(* Logix 5000 project; controller PLC_IA vendor 1 type 14 code 15 rev 20.11; software revision 20.05 *)

TASK MainTask (continuous, watchdog 500 ms) : MainProgram

MODULES
   Local : vendor 1 type 14 code 15 (SoftLogixController 1, rev 20.11)
END_MODULES

VAR_GLOBAL   (* controller tags *)
   ATRASO_SENSOR : REAL := 1000.0;
   CONST_TEMPO : REAL := 15.0;
   DELTA_T : REAL := 0.01;
   ERRO : REAL := 3.9972687;
   FATOR_CONSUMO : REAL := 100.0;
   FLUXO_VAPOR : REAL := 90.0;
   FUZZY_LOOP : FBD_TIMER := (TimerEnable := 1, PRE := 40, ACC := 20, EN := 1, TT := 1);
   FUZZY_ON : BOOL := 1;
   KP : REAL := 3.0;
   KP_MANUAL : REAL := 7.0;
   KP_MAX : REAL := 10.0;
   KP_MIN : REAL := 3.0;
   LIGA_SISTEMA : BOOL := 1;
   MV : REAL := 53.90078;
   P_MAX : REAL := 250.0;
   PV : REAL := 171.15842;
   SP : REAL := 175.0;
   T_AMOST_PID : REAL := 50.0;
   T_LOOP_SISTEMA : REAL := 10.0;
   TAU : REAL := 1.5;
   TD : REAL := 4.274473;
   TD_MANUAL : REAL := 1.0;
   TD_MAX : REAL := 5.0;
   TD_MIN : REAL := 1.0;
   TI : REAL := 5.0;
   TI_INV : REAL := 0.22324193;
   TI_MANUAL : REAL := 3.0;
   TI_MAX : REAL := 5.0;
   TI_MIN : REAL := 0.5;
   VAZAMENTO : REAL;
END_VAR

PROGRAM FUZZY   (* main routine PRINCIPAL *)
VAR
   ACC_DERIVADA : REAL := 0.7598929;
   ACC_DESVIOS_QUADRADO : REAL := 0.0010012466;
   ACC_ERRO : REAL;
   AMOSTRAGEM : FBD_TIMER := (TimerEnable := 1, PRE := 20);
   BUFFER_CIRCULAR : BOOL := 1;
   CONTAGEM : DINT := 46;
   DERIVADA_ALTA : REAL := 0.00604254;
   DERIVADA_BAIXA : REAL := 0.0015563883;
   DERIVADA_FILTRADA : REAL := 0.0023156737;
   DERIVADA_MEDIA : REAL := 0.0037994643;
   DERIVADAS : REAL[5] := ([2] := 0.008644867, [4] := 0.008800507);
   DESVIO : REAL := -0.0014837906;
   DESVIO_PADRAO : REAL := 0.002243076;
   ERRO_ALTO : REAL := 17.5;
   ERRO_ANTERIOR : REAL := 3.9972687;
   ERRO_BAIXO : REAL := 0.17500001;
   ERRO_FILTRADO : REAL := 4.1489806;
   ERRO_MEDIO : REAL := 1.75;
   ERROS : REAL[5] := ([0] := 3.9972687, [1] := 4.346176, [2] := 4.173279, [3] := 4.173279, [4] := 3.9972687);
   EXECUCAO : DINT;
   FILTRAGEM : FBD_TIMER := (TimerEnable := 1, PRE := 20, EN := 1, TT := 1);
   FUZZ_KP : REAL[3] := ([0] := 0.43700165, [2] := 0.1552568);
   FUZZ_TD : REAL[3] := ([0] := 0.1552568, [1] := 0.4403919, [2] := 0.5596081);
   FUZZ_TI : REAL[3] := ([0] := 0.43700165, [1] := 0.8447432, [2] := 0.5596081);
   FUZZY_TIME : REAL := 40.0;
   KP_ALTO : REAL := 10.0;
   KP_BAIXO : REAL := 3.0;
   KP_MEDIO : REAL := 6.5;
   MENOR_VALOR : REAL;
   PERTI_DERIVADA : REAL[3] := ([1] := 0.4403919, [2] := 0.5596081);
   PERTI_ERRO : REAL[3] := ([1] := 0.8447432, [2] := 0.1552568);
   POSICAO : DINT := 1;
   PRIMEIRA_EXECUCAO : BOOL;
   T_AMOSTRAGEM : FBD_TIMER := (Reset := 1);
   TAMANHO_BUFFER : REAL := 200.0;
   TD_ALTO : REAL := 5.0;
   TD_BAIXO : REAL := 1.0;
   TD_MEDIO : REAL := 3.0;
   TEMPO_AMOSTRAGEM : REAL := 20.0;
   TI_ALTO : REAL := 5.0;
   TI_BAIXO : REAL := 0.5;
   TI_MEDIO : REAL := 2.75;
   TIME_FILTRAGEM : REAL := 20.0;
   ULTIMA_DERIVADA : REAL;
   VARIANCIA : REAL := 5.03139e-06;
   VETOR_DERIVADAS : REAL[201] := ([0] := 0.0037889606, [1] := 0.0020592753, [2] := 0.00418396, [3] := 0.0020858257, [4] := 0.0060199993, [5] := 0.003966878, [6] := 0.0034370932, [7] := 0.005819702, [8] := 0.0041832477, [9] := 0.0057259626, [10] := 0.0025300598, [11] := 0.008794352, [12] := 0.005414327, [13] := 0.004825694, [14] := 0.008985087, [15] := 0.006632945, [16] := 0.007867635, [17] := 0.0036768594, [18] := 0.0064361067, [19] := 0.0027026369, [20] := 0.0034643046, [21] := 0.0013593547, [22] := 0.0011015829, [23] := 0.0010068257, [24] := 0.00049591064, [25] := 0.0017445373, [26] := 0.0017635092, [27] := 0.0010932413, [28] := 0.0035477194, [29] := 0.0020349121, [30] := 0.0050069173, [31] := 0.002079061, [32] := 0.0069529214, [33] := 0.0042039487, [34] := 0.00426946, [35] := 0.005052897, [36] := 0.0044214376, [37] := 0.0038611856, [38] := 0.0016247558, [39] := 0.0046980795, [40] := 0.0026897178, [41] := 0.0025284833, [42] := 0.0047458396, [43] := 0.0031422423, [44] := 0.0050496925, [45] := 0.0023156737, [46] := 0.00046005248, [47] := 0.00038441975, [48] := 0.00032608034, [49] := 0.00015319824, [50] := 0.0007211812, [51] := 0.00089324947, [52] := 0.0004510498, [53] := 0.002618103, [54] := 0.0012327576, [55] := 0.0043327333, [56] := 0.0018105062, [57] := 0.005733185, [58] := 0.0038183595, [59] := 0.0038228354,
        [60] := 0.0052285767, [61] := 0.0037962343, [62] := 0.0052091475, [63] := 0.0023093158, [64] := 0.006299642, [65] := 0.0037178549, [66] := 0.0037252808, [67] := 0.0050693764, [68] := 0.0036811319, [69] := 0.005033366, [70] := 0.0022351076, [71] := 0.006123454, [72] := 0.003578135, [73] := 0.0036023457, [74] := 0.004944407, [75] := 0.0035803223, [76] := 0.00487381, [77] := 0.002181193, [78] := 0.0059391274, [79] := 0.0034865316, [80] := 0.0034903463, [81] := 0.0047751362, [82] := 0.0034667968, [83] := 0.004758555, [84] := 0.002109375, [85] := 0.0057554627, [86] := 0.0033972675, [87] := 0.0034038797, [88] := 0.004633484, [89] := 0.003364156, [90] := 0.00460083, [91] := 0.0020432028, [92] := 0.0055985004, [93] := 0.0032713318, [94] := 0.0032933552, [95] := 0.0045218403, [96] := 0.0032740275, [97] := 0.004457957, [98] := 0.0019950867, [99] := 0.0054330444, [100] := 0.0031900024, [101] := 0.0031932069, [102] := 0.004369812, [103] := 0.0031721496, [104] := 0.004355367, [105] := 0.0019306437, [106] := 0.0052687074, [107] := 0.0031103517, [108] := 0.003116099, [109] := 0.004243113, [110] := 0.0030804952, [111] := 0.0042140707, [112] := 0.0018713379, [113] := 0.005128072, [114] := 0.002996877, [115] := 0.0030169168, [116] := 0.0041429647, [117] := 0.0029994203, [118] := 0.0040854393, [119] := 0.0018282572,
        [120] := 0.004979502, [121] := 0.002924245, [122] := 0.0029269918, [123] := 0.004005992, [124] := 0.002907969, [125] := 0.0039934795, [126] := 0.0017700704, [127] := 0.0044295248, [128] := 0.0021709695, [129] := 0.0025767009, [130] := 0.0014201864, [131] := 0.0017451985, [132] := 0.0012846374, [133] := 0.00026168823, [134] := 0.0024367778, [135] := 0.0021867373, [136] := 0.0017131043, [137] := 0.0052009076, [138] := 0.0030574545, [139] := 0.006877899, [140] := 0.0029870605, [141] := 0.009012044, [142] := 0.005469309, [143] := 0.0057130945, [144] := 0.0072477725, [145] := 0.0054625957, [146] := 0.007619018, [147] := 0.003203481, [148] := 0.009398296, [149] := 0.005638784, [150] := 0.005854645, [151] := 0.007651062, [152] := 0.0056430562, [153] := 0.008111725, [154] := 0.0034550477, [155] := 0.009210052, [156] := 0.0057525635, [157] := 0.0058767702, [158] := 0.008184764, [159] := 0.005391744, [160] := 0.00840266, [161] := 0.003948822, [162] := 0.008733826, [163] := 0.004367625, [164] := 0.005135396, [165] := 0.0042689512, [166] := 0.0032692973, [167] := 0.0043944293, [168] := 0.0018687438, [169] := 0.006122894, [170] := 0.004126994, [171] := 0.0038800559, [172] := 0.0067077638, [173] := 0.004504191, [174] := 0.007554728, [175] := 0.0033129374, [176] := 0.008668976, [177] := 0.004777832, [178] := 0.0053255716, [179] := 0.0052858484,
        [180] := 0.004243876, [181] := 0.0037680052, [182] := 0.0018651835, [183] := 0.0036832173, [184] := 0.0015258789, [185] := 0.0017882792, [186] := 0.000923818, [187] := 0.0010198465, [188] := 0.00053400674, [189] := 0.00016108195, [190] := 0.0007420858, [191] := 0.00032419842, [192] := 0.00037216189, [193] := 0.0015240987, [194] := 0.0007048544, [195] := 0.0016716511, [196] := 0.0009288025, [197] := 0.0025672913, [198] := 0.0018614196, [199] := 0.0015527343, [200] := 0.03885905);
   VETOR_DESVIOS : REAL[201] := ([0] := 2.9573382e-06, [1] := 2.5091268e-07, [2] := 1.5205011e-06, [3] := 7.661391e-07, [4] := 1.5119083e-06, [5] := 7.2051694e-06, [6] := 3.784602e-07, [7] := 6.891656e-09, [8] := 5.9700624e-06, [9] := 6.488707e-07, [10] := 5.4367933e-06, [11] := 7.475152e-07, [12] := 2.885194e-05, [13] := 3.9043834e-06, [14] := 1.8993056e-06, [15] := 3.0242056e-05, [16] := 9.806415e-06, [17] := 1.8807697e-05, [18] := 1.8989514e-08, [19] := 8.281695e-06, [20] := 7.388706e-07, [21] := 1.0648864e-08, [22] := 4.88189e-06, [23] := 6.0449424e-06, [24] := 6.505347e-06, [25] := 9.338245e-06, [26] := 3.2610042e-06, [27] := 3.197212e-06, [28] := 6.0241664e-06, [29] := 1.8111357e-10, [30] := 2.3277132e-06, [31] := 2.0372106e-06, [32] := 2.2642676e-06, [33] := 1.1167069e-05, [34] := 3.3333185e-07, [35] := 3.946825e-07, [36] := 1.9304443e-06, [37] := 5.5261563e-07, [38] := 2.8178214e-08, [39] := 4.2948723e-06, [40] := 9.648893e-07, [41] := 1.072789e-06, [42] := 1.4534289e-06, [43] := 9.799563e-07, [44] := 3.9057537e-07, [45] := 1.58615e-06, [46] := 8.007315e-06, [47] := 8.10455e-06, [48] := 8.487863e-06, [49] := 8.782421e-06, [50] := 9.7864795e-06, [51] := 6.4863684e-06, [52] := 5.606348e-06, [53] := 7.79847e-06, [54] := 3.9699964e-07, [55] := 3.997394e-06, [56] := 1.1974279e-06, [57] := 2.023872e-06, [58] := 6.2132062e-06, [59] := 3.2789654e-07,
        [60] := 3.4131332e-07, [61] := 3.900039e-06, [62] := 3.1043325e-07, [63] := 3.865559e-06, [64] := 8.5381527e-07, [65] := 9.403526e-06, [66] := 2.388203e-07, [67] := 2.6127444e-07, [68] := 3.4021562e-06, [69] := 2.2981268e-07, [70] := 3.3539004e-06, [71] := 9.082978e-07, [72] := 8.640061e-06, [73] := 1.610975e-07, [74] := 1.9430595e-07, [75] := 3.144376e-06, [76] := 1.8326233e-07, [77] := 2.9420125e-06, [78] := 9.357414e-07, [79] := 7.683639e-06, [80] := 9.994215e-08, [81] := 9.622623e-08, [82] := 2.4721726e-06, [83] := 6.588723e-08, [84] := 2.3537712e-06, [85] := 1.2501492e-06, [86] := 6.356949e-06, [87] := 2.5232172e-08, [88] := 3.0898907e-08, [89] := 1.9450006e-06, [90] := 2.0357055e-08, [91] := 1.890251e-06, [92] := 1.3742845e-06, [93] := 5.6442605e-06, [94] := 2.4645186e-09, [95] := 5.3044302e-09, [96] := 1.6544536e-06, [97] := 1.5958361e-09, [98] := 1.4656536e-06, [99] := 1.5662874e-06, [100] := 4.6900473e-06, [101] := 7.498061e-09, [102] := 9.312055e-09, [103] := 1.1222714e-06, [104] := 2.2385308e-08, [105] := 1.0286437e-06, [106] := 2.0112932e-06, [107] := 3.609533e-06, [108] := 7.2895325e-08, [109] := 7.4481704e-08, [110] := 6.990904e-07, [111] := 1.1010914e-07, [112] := 6.207139e-07, [113] := 2.427668e-06, [114] := 2.845061e-06, [115] := 2.0363854e-07, [116] := 1.8261623e-07, [117] := 4.705508e-07, [118] := 1.9731706e-07, [119] := 4.108834e-07,
        [120] := 2.5830077e-06, [121] := 2.4127462e-06, [122] := 2.441865e-07, [123] := 2.1766195e-07, [124] := 3.7180462e-07, [125] := 2.0217527e-07, [126] := 4.2309293e-07, [127] := 2.3991495e-06, [128] := 1.3035926e-06, [129] := 1.1903454e-06, [130] := 4.0863705e-07, [131] := 3.158271e-06, [132] := 1.917442e-06, [133] := 3.253678e-06, [134] := 7.737029e-06, [135] := 2.980862e-07, [136] := 5.727842e-07, [137] := 1.3515066e-06, [138] := 5.4450447e-06, [139] := 7.169536e-08, [140] := 1.6864713e-05, [141] := 6.5627745e-08, [142] := 3.9622384e-05, [143] := 7.695371e-06, [144] := 9.224776e-06, [145] := 2.0757028e-05, [146] := 7.797909e-06, [147] := 2.4361989e-05, [148] := 2.8252762e-07, [149] := 4.498373e-05, [150] := 8.652641e-06, [151] := 9.921689e-06, [152] := 2.4187766e-05, [153] := 8.438927e-06, [154] := 2.8561488e-05, [155] := 4.6599374e-07, [156] := 4.1015617e-05, [157] := 8.573145e-06, [158] := 9.207904e-06, [159] := 2.8160855e-05, [160] := 6.2536906e-06, [161] := 3.0007364e-05, [162] := 1.0253484e-06, [163] := 3.3237407e-05, [164] := 1.9191352e-06, [165] := 4.571872e-06, [166] := 1.575745e-06, [167] := 6.3512125e-08, [168] := 1.8560517e-06, [169] := 1.3580159e-06, [170] := 9.41174e-06, [171] := 1.1200739e-06, [172] := 6.4198497e-07, [173] := 1.2957162e-05, [174] := 1.9173199e-06, [175] := 1.9393981e-05, [176] := 2.3088429e-08, [177] := 2.995802e-05, [178] := 2.4483259e-06, [179] := 4.3870746e-06,
        [180] := 4.1300164e-06, [181] := 9.595819e-07, [182] := 2.411631e-07, [183] := 2.0017692e-06, [184] := 1.5463954e-07, [185] := 3.1172626e-06, [186] := 2.2611748e-06, [187] := 5.612499e-06, [188] := 5.1435136e-06, [189] := 7.565125e-06, [190] := 9.723186e-06, [191] := 6.414435e-06, [192] := 8.680194e-06, [193] := 8.363685e-06, [194] := 3.0417334e-06, [195] := 6.5379736e-06, [196] := 2.536733e-06, [197] := 5.449436e-06, [198] := 4.911451e-07, [199] := 1.9887643e-06);
   VETOR_ERRO : REAL[201];
END_VAR

ROUTINE FUZZY   (* structured text *)
   ////////////////////////////////////////////////////////////////////////////////////////
   //						FILTRAGEM DAS VARIAVES DE ENTRADA
   ////////////////////////////////////////////////////////////////////////////////////////
   
   
   
   //TIMER DE FILTRAGEM
   TONR(FILTRAGEM);
   TIME_FILTRAGEM			:= T_LOOP_SISTEMA*2;
   FILTRAGEM.PRE 			:= TIME_FILTRAGEM;
   FILTRAGEM.ENABLEIN 		:= 1;
   FILTRAGEM.RESET 		:= 0;
   FILTRAGEM.TIMERENABLE	:= 1;
   
   
   //DISPARO DO TIMER
   IF FILTRAGEM.DN THEN
   
   	//RESETA O TIMER
   	FILTRAGEM.RESET := 1;
   
   	//SALVA O ERRO ABSOLUTO ATUAL
   	ERROS[POSICAO]:= ABS(ERRO);
   
   	//SALVA A DERIVADA ABSOLUTA ATUAL
   	DERIVADAS[POSICAO] := ABS((ERROS[POSICAO] - ERRO_ANTERIOR)/TIME_FILTRAGEM);
   
   	//SALVA O ULTIMO ERRO
   	ERRO_ANTERIOR := ERROS[POSICAO];
   
   	//NAO DEIXA TIRAR A MEDIA PONDERADA ENQUANTO O BUFFER NAO ESTA COMPLETAMENTE CHEIO
   	IF NOT(PRIMEIRA_EXECUCAO) THEN
   
   		//ERRO DE ENTRADA DO FUZZIFICADOR
   		ERRO_FILTRADO := (ERROS[(POSICAO) MOD 5]*5 + ERROS[(POSICAO+1) MOD 5]*4 + ERROS[(POSICAO+2) MOD 5]*3
   					+ ERROS[(POSICAO+3) MOD 5]*2 + ERROS[(POSICAO+4) MOD 5])/15;
   
   		//DERIVADA DE ENTRADA DO FUZZIFICADOR
   		DERIVADA_FILTRADA := (DERIVADAS[(POSICAO) MOD 5]*5 + DERIVADAS[(POSICAO+1) MOD 5]*4 + DERIVADAS[(POSICAO+2) MOD 5]*3
   					+ DERIVADAS[(POSICAO+3) MOD 5]*2 + DERIVADAS[(POSICAO+4) MOD 5])/15;
   	ELSE
   
   		//CONTA A QUANTIDADE DE POSICOES CHEIAS NO BUFFER
   		EXECUCAO := EXECUCAO + 1;
   
   		//SE ENCHEU FLIPA O BIT QUE DEIXA TIRAR A MEDIA
   		IF EXECUCAO > 4 THEN
   			EXECUCAO 		 	:= 0;
   			PRIMEIRA_EXECUCAO 	:= 0;
   		END_IF;
   
   	END_IF;
   
   
   	//INCREMENTA O BUFFER CIRCULAR
   	POSICAO := (POSICAO + 1) MOD 5;
   
   END_IF;
   
   
   
   
   ////////////////////////////////////////////////////////////////////////////////////////
   //		DEFININDO OS REFERENCIAIS DE ERRO
   
   ERRO_BAIXO := 0.001*SP;
   ERRO_MEDIO := 0.05*SP;
   ERRO_ALTO  := 0.15*SP;
   
   
   ////////////////////////////////////////////////////////////////////////////////////////
   //		ANALIZANDO AS ESTATISTICAS DAS ULTIMAS 200 VARIACOES DO ERRO (DERIVADA)
   
   
   //TIMER DE AMOSTRAGEM
   TONR(AMOSTRAGEM);
   TEMPO_AMOSTRAGEM		:= T_LOOP_SISTEMA*2;
   AMOSTRAGEM.PRE 			:= TEMPO_AMOSTRAGEM;
   AMOSTRAGEM.ENABLEIN 	:= 1;
   AMOSTRAGEM.TIMERENABLE 	:= 1;
   AMOSTRAGEM.RESET 		:= 0;
   
   IF AMOSTRAGEM.DN THEN
   
   	AMOSTRAGEM.RESET 		:= 1;
   	AMOSTRAGEM.TIMERENABLE 	:= 0;
   
   	//SE AUMENTAR MUITO ATRASA A RESPOSTA
   	TAMANHO_BUFFER := 200;
   
   	//LIGA O BUFFER CIRCULAR
   	IF BUFFER_CIRCULAR THEN
   
   		//RETIRA O ULTIMO VALOR DO VETOR DE DERIVADAS
   		ACC_DERIVADA := ACC_DERIVADA - VETOR_DERIVADAS[CONTAGEM];
   
   		//RETIRA O ULTIMO VALOR DO VETOR DE DESVIOS
   		ACC_DESVIOS_QUADRADO := ACC_DESVIOS_QUADRADO - VETOR_DESVIOS[CONTAGEM];
   
   	END_IF;
   
   	//ACUMULA OS K-ULTIMOS VALORES
   	ACC_DERIVADA:= ACC_DERIVADA + DERIVADA_FILTRADA;
   	ACC_DESVIOS_QUADRADO := ACC_DESVIOS_QUADRADO + DESVIO*DESVIO;
   
   	//SALVA A ULTIMA DERIVADA NO VETOR
   	VETOR_DERIVADAS[CONTAGEM] :=  DERIVADA_FILTRADA;
   
   	//SALVA O ULTIMO DESVIO NO VETOR
   	VETOR_DESVIOS[CONTAGEM] :=  DESVIO*DESVIO;
   
   	//INCREMENTA A CONTAGEM DE DERIVADAS
   	CONTAGEM := CONTAGEM + 1;
   
   	//SE A JANELA ENCHEU, LIGA O BUFFER CIRCULAR E VOLTA AO SEU INICIO
   	IF CONTAGEM > TAMANHO_BUFFER-1 THEN
   		BUFFER_CIRCULAR :=1;
   		CONTAGEM := 0;
   	END_IF;
   
   ////////////////////////////////////////////////////////////////////////////////////////
   //		DEFININDO OS REFERENCIAIS DA DERIVADA DO ERRO
   
   	//DERIVADA MEDIA (VARIAVEL DE REFERENCIA)
   	DERIVADA_MEDIA := ACC_DERIVADA/TAMANHO_BUFFER;
   
   	//DESVIO
   	DESVIO := DERIVADA_FILTRADA - DERIVADA_MEDIA;
   
   	//VARIANCIA COM UM GRAU DE LIBERDADE
   	VARIANCIA := ACC_DESVIOS_QUADRADO/(TAMANHO_BUFFER-1);
   
   	//DESVIO PADRAO
   	DESVIO_PADRAO := SQRT(VARIANCIA);
   
   	//VARIAVEIS DE REFERENCIA RESTANTES
   	DERIVADA_BAIXA := DERIVADA_MEDIA - DESVIO_PADRAO;
   	IF DERIVADA_BAIXA < 0 THEN
   		DERIVADA_BAIXA := 0;
   	END_IF;
   	DERIVADA_ALTA  := DERIVADA_MEDIA + DESVIO_PADRAO;
   
   END_IF;
   
   
   ////////////////////////////////////////////////////////////////////////////////////////
   //							CONTROLE DO ALGORITMO FUZZY
   ////////////////////////////////////////////////////////////////////////////////////////
   
   //TEMPO DE LOOP_FUZZY EM MILISSEGUNDOS
   //FUZZY_TIME := (TEMPO_AMOSTRAGEM*TAMANHO_BUFFER)/4;
   FUZZY_TIME := TEMPO_AMOSTRAGEM*2;
   
   //LIGA FUZZY
   IF FUZZY_ON THEN
   
   	//TIMER DE LOOP FUZZY
   	TONR(FUZZY_LOOP);
   	FUZZY_LOOP.PRE 			:= FUZZY_TIME;
   	FUZZY_LOOP.ENABLEIN 	:= 1;
   	FUZZY_LOOP.TIMERENABLE 	:= 1;
   	FUZZY_LOOP.RESET 		:= 0;
   
   ELSE
   	//RESET DO TEMPORIZADOR
   	FUZZY_LOOP.ENABLEIN 	:= 0;
   	FUZZY_LOOP.TIMERENABLE 	:= 0;
   	FUZZY_LOOP.RESET 		:= 1;
   	FUZZY_LOOP.DN			:= 0;
   
   	//RESET DAS VARIAVEIS DA MEDIA MOVEL
   	BUFFER_CIRCULAR			:= 0;
   	ACC_DERIVADA			:= 0;
   	ACC_DESVIOS_QUADRADO	:= 0;
   	CONTAGEM				:= 0;
   
   
   	//DESLIGA A AMOSTRAGEM ESTATISTICA
   	T_AMOSTRAGEM.TIMERENABLE 	:= 0;
   	T_AMOSTRAGEM.RESET 			:= 1;
   
   	//RETORNA AS VARIAVEIS SINTONIZADAS MANUALMENTE
   	KP := KP_MANUAL;
   	TI := TI_MANUAL;
   	TD := TD_MANUAL;
   
   	//RESET DA FILTRAGEM
   	POSICAO				:= 0;
   	ERRO_FILTRADO		:= 0;
   	DERIVADA_FILTRADA	:= 0;
   	PRIMEIRA_EXECUCAO 	:= 1;
   	EXECUCAO 		 	:= 0;
   
   
   END_IF;
   
   
   
   ////////////////////////////////////////////////////////////////////////////////////////
   //							INICIO DO ALGORITMO FUZZY
   ////////////////////////////////////////////////////////////////////////////////////////
   
   //TESTA SE O TIMER DE LOOP DISPAROU
   IF FUZZY_LOOP.DN THEN;
   
   
   ///////////////////////////////////////////////////////////////////////////////
   //			CALCULO DO VETOR DE PERTINENCIA DO ERRO
   
   	//CERTEZA DE QUE O ERRO EH BAIXO
   	IF ERRO_FILTRADO <= ERRO_BAIXO THEN
   		PERTI_ERRO[0] := 1;	//ERRO BAIXO
   		PERTI_ERRO[1] := 0;	//ERRO MEDIO
   		PERTI_ERRO[2] := 0;	//ERRO ALTO
   	ELSE
   
   		//CERTEZA DE QUE O ERRO EH ALTO
   		IF ERRO_FILTRADO >= ERRO_ALTO THEN
   			PERTI_ERRO[0] := 0;	//ERRO BAIXO
   			PERTI_ERRO[1] := 0;	//ERRO MEDIO
   			PERTI_ERRO[2] := 1;	//ERRO ALTO
   		ELSE
   
   			//MEIO TERMO
   			IF ERRO_FILTRADO < ERRO_MEDIO THEN
   
   				//SO PRA GARANTIR QUE NAO VAI DAR ERRO DE DIVISAO POR ZERO
   				IF ERRO_MEDIO <> ERRO_BAIXO THEN
   
   					//VAMOS CALCULAR PRIMEIRO O ERRO MEDIO
   					PERTI_ERRO[1] := (ERRO_FILTRADO-ERRO_BAIXO)/(ERRO_MEDIO-ERRO_BAIXO);
   
   				END_IF;
   
   				//ERRO BAIXO
   				PERTI_ERRO[0] := 1 - PERTI_ERRO[1];
   
   				//ERRO ALTO
   				PERTI_ERRO[2] := 0;
   
   			ELSE
   
   				//SO PRA GARANTIR QUE NAO VAI DAR ERRO DE DIVISAO POR ZERO
   				IF ERRO_MEDIO <> ERRO_ALTO THEN
   
   					//VAMOS CALCULAR PRIMEIRO O ERRO ALTO
   					PERTI_ERRO[2] := (ERRO_FILTRADO- ERRO_MEDIO)/(ERRO_ALTO-ERRO_MEDIO);
   
   				END_IF;
   
   				//PERTINENCIA DO ERRO MEDIO
   				PERTI_ERRO[1] := 1 - PERTI_ERRO[2];
   
   				//PERTINENCIA DO ERRO BAIXO
   				PERTI_ERRO[0] := 0;
   
   			END_IF;	//FIM IF MEIO TERMO
   		END_IF; //FIM IF ALTO
   	END_IF; //FIM IF BAIXO
   
   
   
   ///////////////////////////////////////////////////////////
   //		CALCULO DO VETOR DE PERTINENCIA DA DERIVADA
   
   	//CERTEZA DE QUE A DERIVADA EH BAIXA
   	IF DERIVADA_FILTRADA <= DERIVADA_BAIXA THEN
   		PERTI_DERIVADA[0] := 1;	//DERIVADA BAIXA
   		PERTI_DERIVADA[1] := 0;	//DERIVADA MEDIA
   		PERTI_DERIVADA[2] := 0;	//DERIVADA ALTA
   	ELSE
   
   		//CERTEZA DE QUE A DERIVADA EH ALTA
   		IF DERIVADA_FILTRADA >= DERIVADA_ALTA THEN
   			PERTI_DERIVADA[0] := 0;	//DERIVADA BAIXA
   			PERTI_DERIVADA[1] := 0;	//DERIVADA MEDIA
   			PERTI_DERIVADA[2] := 1;	//DERIVADA ALTA
   		ELSE
   
   			//MEIO TERMO
   			IF DERIVADA_FILTRADA < DERIVADA_MEDIA THEN
   
   				//SO PRA GARANTIR QUE NAO VAI DAR ERRO DE DIVISAO POR ZERO
   				IF DERIVADA_MEDIA <> DERIVADA_BAIXA THEN
   
   					//VAMOS CALCULAR PRIMEIRO A PERTINENCIA DA DERIVADA MEDIA
   					PERTI_DERIVADA[1] := (DERIVADA_FILTRADA-DERIVADA_BAIXA)/(DERIVADA_MEDIA-DERIVADA_BAIXA);
   
   				END_IF;
   
   				//PERTINENCIA DA DERIVADA BAIXA
   				PERTI_DERIVADA[0] := 1 - PERTI_DERIVADA[1];
   
   				//PERTINENCIA DA DERIVADA ALTA
   				PERTI_DERIVADA[2] := 0;
   
   			ELSE
   
   				//SO PRA GARANTIR QUE NAO VAI DAR ERRO DE DIVISAO POR ZERO
   				IF DERIVADA_MEDIA <> DERIVADA_ALTA THEN
   
   					//VAMOS CALCULAR PRIMEIRO A DERIVADA ALTA
   					PERTI_DERIVADA[2] := (DERIVADA_FILTRADA-DERIVADA_MEDIA)/(DERIVADA_ALTA-DERIVADA_MEDIA);
   
   				END_IF;
   
   				//PERTINENCIA DA DERIVADA MEDIA
   				PERTI_DERIVADA[1] := 1 - PERTI_DERIVADA[2];
   
   				//PERTINENCIA DA DERIVADA BAIXA
   				PERTI_DERIVADA[0] := 0;
   
   			END_IF;	//FIM IF MEIO TERMO
   		END_IF; //FIM IF ALTA
   	END_IF; //FIM IF BAIXA
   
   
   
   ///////////////////////////////////////////////////////////////////////////////
   //					CALCULANDO AS INFERENCIAS FUZZY
   //   	(AQUI EH ONDE A MAQUINA APRENDE O PENSAMENTO DO PROGRAMADOR)
   ///////////////////////////////////////////////////////////////////////////////
   
   
   
   //////////////////////////////////////////////////////////////////////////////
   //							INFERENCIAS DO KP
   
   	//	SE O ERRO EH BAIXO ENTAO DIMINUI O KP...
   	//	=> EVITA OSCILACOES
   	FUZZ_KP[0] := PERTI_ERRO[0];
   
   
   	//	SE O ERRO EH BAIXO E A TI EH ALTA ENTAO DIMINUI O KP...
   	//	=> DEIXA O TRABALHO PRO TI
   	FUZZ_KP[0] := PERTI_ERRO[0];
   
   	IF FUZZ_TI[2] < FUZZ_KP[0] THEN
   		FUZZ_KP[0] := FUZZ_TI[2];
   	END_IF;
   
   
   	//	SE O ERRO EH MEDIO ENTAO O KP EH MEDIO...
   	//	=> CORRECAO MODERADA
   	FUZZ_KP[1] := PERTI_ERRO[1];
   
   
   	//	SE O ERRO EH MEDIO E O TI EH BAIXO E A DERIVADA EH BAIXA ENTAO O KP EH MEDIO...
   	//	=> CORRECAO MODERADA
   	FUZZ_KP[1] := PERTI_ERRO[1];
   
   	IF FUZZ_TI[0] < FUZZ_KP[1] THEN
   		FUZZ_KP[1] := FUZZ_TI[0];
   	END_IF;
   
   
   	//	SE O ERRO EH ALTO ENTAO AUMENTA O KP...
   	//	=> CORRECAO RAPIDA SEM AUMENTAR AS OSCILACOES E EVITANDO OVERSHOOTING
   	FUZZ_KP[2] := PERTI_ERRO[2];
   
   
   
   //////////////////////////////////////////////////////////////////////////////
   //							INFERENCIAS DO TI
   
   	//	SE O ERRO EH ALTO ENTAO DIMINUI O TI...
   	//	=> ACUMULACAO RAPIDA PARA CORRECAO RAPIDA
   	FUZZ_TI[0] := PERTI_ERRO[2];
   
   	//	SE (O ERRO EH BAIXO OU MEDIO) E O KP EH BAIXO ENTAO DIMUNUI O TI...
   	//	=> ACUMULACAO LENTA PARA EVITAR OVERSHOOTING
   	FUZZ_TI[0] := PERTI_ERRO[0];
   	IF FUZZ_TI[0] < PERTI_ERRO[1] THEN
   		FUZZ_TI[0] := PERTI_ERRO[1];
   	END_IF;
   	IF FUZZ_TI[0] < FUZZ_KP[0] THEN
   		FUZZ_TI[0] := FUZZ_KP[0];
   	END_IF;
   
   
   	//	SE O ERRO EH MEDIO ENTAO O TI EH MEDIO...
   	//	=> CORRECAO SUAVE E ESTAVEL
   	FUZZ_TI[1] := PERTI_ERRO[1];
   
   
   	//	SE O ERRO EH BAIXO E A DERIVADA EH ALTA ENTAO AUMENTA O TI...
   	//	=> ACUMULACAO LENTA PARA EVITAR OVERSHOOTING
   	FUZZ_TI[2] := PERTI_ERRO[0];
   	IF FUZZ_TI[2] < PERTI_DERIVADA[2] THEN
   		FUZZ_TI[2] := PERTI_DERIVADA[2];
   	END_IF;
   
   
   
   //////////////////////////////////////////////////////////////////////////////
   //							INFERENCIAS DO TD
   
   	//	SE O ERRO EH ALTO ENTAO DIMINUI O TD...
   	//	=> DERIVATIVO MINIMO PARA EVITAR AMORTECER A CORRECAO RAPIDA
   	FUZZ_TD[0] := PERTI_ERRO[2];
   
   	//	SE A DERIVADA EH BAIXA ENTAO DIMINUI O TD...
   	//	=> DIMINUI O AMORTECIMENTO PARA O TI RECUPERAR O ERRO MINIMO
   	FUZZ_TD[0] := PERTI_DERIVADA[0];
   
   
   	//	SE DERIVADA EH MEDIA ENTAO O TD EH MEDIO...
   	//	=> AMORTECIMENTO MODERADO
   	FUZZ_TD[1] := PERTI_DERIVADA[1];
   
   
   	//	SE A DERIVADA EH ALTA ENTAO AUMENTA O TD...
   	//	=> FORTE AMORTECIMENTO PARA PEQUENAS VARIACOES
   	FUZZ_TD[2] := PERTI_DERIVADA[2];
   
   
   
   ///////////////////////////////////////////////////////////////////////////////
   //					DEFUZZYFICACAO DAS INFERENCIAS
   //   			(AQUI EH ONDE A MAQUINA TOMA UMA DECISAO)
   ///////////////////////////////////////////////////////////////////////////////
   
   
   //////////////////////////////////////////////////////////////////////////////
   //						VARIAVEIS DE DEFUZIFICACAO
   
   	KP_BAIXO 	:= KP_MIN;
   	KP_MEDIO 	:= (KP_MIN + KP_MAX)/2;
   	KP_ALTO		:= KP_MAX;
   
   	TI_BAIXO 	:= TI_MIN;
   	TI_MEDIO 	:= (TI_MIN + TI_MAX)/2;
   	TI_ALTO		:= TI_MAX;
   
   	TD_BAIXO 	:= TD_MIN;
   	TD_MEDIO 	:= (TD_MIN + TD_MAX)/2;
   	TD_ALTO		:= TD_MAX;
   
   
   //////////////////////////////////////////////////////////////////////////////
   //							CALCULO DAS SAIDAS
   //	(COMBINACAO LINEAR DOS VETORES DE INFERENCA E AS VARIAVEIS FUZZY)
   
   	//KP RESULTANTE
   	KP := FUZZ_KP[0]*KP_BAIXO +	FUZZ_KP[1]*KP_MEDIO + FUZZ_KP[2]*KP_ALTO;
   
   	IF KP < KP_BAIXO THEN
   		KP := KP_BAIXO;
   	END_IF;
   	IF KP > KP_ALTO THEN
   		KP := KP_ALTO;
   	END_IF;
   
   	//TI RESULTANTE
   	TI := FUZZ_TI[0]*TI_BAIXO +	FUZZ_TI[1]*TI_MEDIO + FUZZ_TI[2]*TI_ALTO;
   
   	IF TI < TI_BAIXO THEN
   		TI := TI_BAIXO;
   	END_IF;
   	IF TI > TI_ALTO THEN
   		TI := TI_ALTO;
   	END_IF;
   
   	//TD RESULTANTE
   	TD := FUZZ_TD[0]*TD_BAIXO +	FUZZ_TD[1]*TD_MEDIO + FUZZ_TD[2]*TD_ALTO;
   
   	IF TD < TD_BAIXO THEN
   		TD := TD_BAIXO;
   	END_IF;
   	IF TD > TD_ALTO THEN
   		TD := TD_ALTO;
   	END_IF;
   
   
   //////////////////////////////////////////////////////////////////////////////
   //									FIM!
   
   	//REINICIA O TIMER
   	FUZZY_LOOP.RESET := 1;
   
   END_IF;
   
   
   
   
   
   
   
   
   
   
   
END_ROUTINE

ROUTINE PRINCIPAL   (* ladder *)
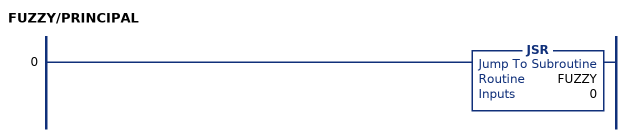
   0: JSR(FUZZY,0);
END_ROUTINE
END_PROGRAM

PROGRAM MainProgram   (* main routine MainRoutine *)
VAR
   ABERTURA_VALVULA : REAL := 31.59636;
   ACC_MEDIA_MOVEL : REAL := 8557.921;
   ALEATORIO : REAL := 0.4097222;
   ARMAZENA : BOOL;
   AUX : REAL := 187.0;
   BUFFER_CIRCULAR : BOOL := 1;
   CALCULA_ALEATORIOS : BOOL := 1;
   CONSUMINDO : REAL := 1.0;
   CONSUMIR : BOOL;
   CONSUMO_ALEATORIO : REAL := 12292.666;
   CONTAGEM : DINT := 30;
   DERIVADA : REAL := -3.1137085;
   DISSIPACAO : REAL := 2.1960408e-05;
   ERRO_ANTERIOR : REAL := 3.8415833;
   INTEGRAL : REAL := 100.0;
   P_ENTRADA : REAL := 131.67386;
   P_SAIDA : REAL := 173.98529;
   P_T0 : REAL := 173.98529;
   SEED : REAL := 177.0;
   T_MEDIA_MOVEL : FBD_TIMER;
   TAMANHO_BUFFER : DINT := 50;
   TEMPO_CONSUMINDO : FBD_TIMER := (PRE := 2674, Reset := 1);
   TEMPO_LOOP_PID : FBD_TIMER := (TimerEnable := 1, PRE := 50);
   TEMPO_LOOP_SISTEMA : FBD_TIMER := (TimerEnable := 1, PRE := 10);
   TEMPO_MEDIA_MOVEL : FBD_TIMER := (TimerEnable := 1, PRE := 20, ACC := 10, EN := 1, TT := 1);
   TEMPO_SEM_CONSUMO : FBD_TIMER := (TimerEnable := 1, PRE := 1444, ACC := 810, EN := 1, TT := 1);
   TIME_PID : REAL := 0.05;
   ULTIMA_ADD : REAL;
   VETOR_VALORES : REAL[1000] := ([0] := 167.13223, [1] := 166.23515, [2] := 166.47327, [3] := 166.94592, [4] := 167.18048, [5] := 167.41386, [6] := 167.8771, [7] := 168.10698, [8] := 168.3357, [9] := 168.78966, [10] := 169.01492, [11] := 169.51672, [12] := 170.51031, [13] := 171.00215, [14] := 171.4907, [15] := 172.45808, [16] := 171.5366, [17] := 170.62128, [18] := 170.30583, [19] := 170.14967, [20] := 170.64392, [21] := 171.62254, [22] := 172.10696, [23] := 172.58817, [24] := 173.54094, [25] := 173.72496, [26] := 173.90775, [27] := 174.843, [28] := 174.55519, [29] := 174.26929, [30] := 170.95303, [31] := 171.16731, [32] := 171.59259, [33] := 171.8036, [34] := 172.01353, [35] := 172.43019, [36] := 172.63692, [37] := 172.84259, [38] := 172.9417, [39] := 172.83673, [40] := 173.04138, [41] := 173.44753, [42] := 173.64903, [43] := 173.8495, [44] := 174.24736, [45] := 172.81616, [46] := 171.39232, [47] := 171.03271, [48] := 170.8543, [49] := 169.44048, [50] := 172.78691, [51] := 172.93922, [52] := 173.01941, [53] := 173.05922, [54] := 173.23488, [55] := 173.5837, [56] := 173.75685, [57] := 173.92918, [58] := 174.2714, [59] := 174.35896,
        [60] := 174.44612, [61] := 174.78339, [62] := 174.9508, [63] := 175.11743, [64] := 175.44176, [65] := 175.5995, [66] := 175.66508, [67] := 175.85965, [68] := 175.98831, [69] := 176.11635, [70] := 176.27974, [71] := 176.32275, [72] := 176.36557, [73] := 176.40746, [74] := 176.42824, [75] := 150.98894, [76] := 151.64899, [77] := 152.95592, [78] := 153.60286, [79] := 154.24548, [80] := 155.5179, [81] := 156.14775, [82] := 156.7734, [83] := 158.01224, [84] := 158.62546, [85] := 159.22095, [86] := 160.4002, [87] := 160.98402, [88] := 161.564, [89] := 162.7125, [90] := 163.28108, [91] := 163.84592, [92] := 164.96445, [93] := 165.5182, [94] := 166.0683, [95] := 167.15765, [96] := 167.69695, [97] := 168.23268, [98] := 169.2936, [99] := 169.81882);
END_VAR

ROUTINE MainRoutine   (* ladder *)
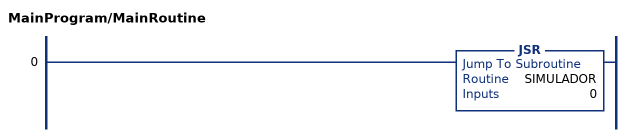
   0: JSR(SIMULADOR,0);
END_ROUTINE

ROUTINE SIMULADOR   (* structured text *)
   
   //	PROJETO:	SIMULADOR DE SISTEMA DE PRIMEIRA ORDEM COM CONTROLE PID, CONSUMO E ALGUNS DISTURBIOS
   //	AUTOR:		ENG. LUZENILTON TORRES
   //	DATA:		20/09/2024
   
   
   //DISTURBIOS DO SISTEMA: (VAR:REAL)
   //FLUXO_VAPOR		:= 100;		//FLUXO DE VAPOR DE ENTRADA DE 0 A 100% (SAIDA DA CALDEIRA)
   //VAZAMENTO			:= 0;		//SIMULA UM VAZAMENTO POSTERIOR AUMENTANDO A CONSTANTE DE TEMPO (0 A 100 SEGUNDOS)
   //FATOR_CONSUMO		:= 20;		//CONSUMO DE VAPOR PELOS EQUIPAMENTOS (0 A 100%)
   //ATRASO_SENSOR   	:= 100;		//ATRASO DE RESPOSTA DO SENSOR EM MILISSEGUNDOS
   
   //CONSTANTES DO SISTEMA: (VAR:REAL)
   //CONST_TEMPO 		:= 20;		//CONSTANTE DE TEMPO (EM SEGUNDOS)
   //P_MAX 			:= 250;		//PRESSAO MAXIMA DO SISTEMA
   T_LOOP_SISTEMA		:= 10;		//TEMPO DE LOOP DOS CALCULOS DO SISTEMA
   
   //AJUSTES DO CONTROLADOR: (VAR:REAL)
   //SP					:= 160;		//PRESSAO DESEJADA (PSI)
   //KP					:= 7.5;		//GANHO PROPORCIONAL
   //TI					:= 2.0;		//GANHO INTEGRAL
   //TD					:= 1.2;		//GANHO DERIVATIVO
   
   
   //TIMERS
   TONR(TEMPO_LOOP_SISTEMA);
   TONR(TEMPO_LOOP_PID);
   TONR(TEMPO_SEM_CONSUMO);
   TONR(TEMPO_CONSUMINDO);
   TONR(TEMPO_MEDIA_MOVEL);
   
   /////////////////////////////////////////////////////////////////////////////////////////
   //						SIMULADOR DE SISTEMA DE PRIMEIRA ORDEM
   ////////////////////////////////////////////////////////////////////////////////////////
   
   //PEGA O TEMPO DE LOOP DO SISTEMA E CONVERTE PARA SEGUNDOS
   DELTA_T := T_LOOP_SISTEMA/1000;
   
   //CONSTANTE DE TEMPO
   TAU := (CONST_TEMPO + VAZAMENTO*FATOR_CONSUMO)/T_LOOP_SISTEMA;
   
   //SIMULACAO DO SISTEMA
   IF LIGA_SISTEMA THEN
   
   	TEMPO_LOOP_SISTEMA.PRE			:= T_LOOP_SISTEMA;
   	TEMPO_LOOP_SISTEMA.ENABLEIN 	:= 1;
   	TEMPO_LOOP_SISTEMA.RESET		:= 0;
   	TEMPO_LOOP_SISTEMA.TIMERENABLE	:= 1;
   
   	IF TEMPO_LOOP_SISTEMA.DN THEN
   
   		//PEGA A ABERTURA DA VALVULA (SAIDA DO PID)
   		MV := ABERTURA_VALVULA;
   
   		//CALCULA A PRESSAO DE ENTRADA
   		P_ENTRADA := (MV/100.0)*P_MAX*(LN(FLUXO_VAPOR)/(4.605));
   
   		//EQUACAO DO SISTEMA
   		P_SAIDA := P_T0 + (DELTA_T/TAU)*(P_ENTRADA-P_SAIDA) - DISSIPACAO;
   
   		//ATUALIZA OS INSTANTES
   		P_T0	:= P_SAIDA;
   
   		//DISSIPACAO DE ENERGIA (PRA SIMULAR UNS PEQUENOS VAZAMENTOS E FICAR MAIS REAL):
   		DISSIPACAO := (1/(P_MAX*P_SAIDA+1000))*(LN(FLUXO_VAPOR)/(4.605))*CONSUMINDO; //SIMULA O CONSUMO PELOS EQUIPAMENTOS
   
   		IF P_SAIDA <= 0 THEN
   			P_SAIDA := 0;
   		END_IF;
   
   		TEMPO_LOOP_SISTEMA.RESET := 1;
   
   	END_IF;
   
   ELSE
   
   	//RESET DE VALORES
   	P_SAIDA 					:= 0.0;		//PRESSAO SAIDA
   	P_T0						:= 0.0;		//PRESSAO NO INSTANTE T0
   	MV							:= 0.0;		//ABERTURA DA VALVULA
   	INTEGRAL 					:= 0.0; 	//RESET DA INTEGRAL
   	BUFFER_CIRCULAR				:= 0;		//RESET DO BUFFER CIRCULAR
   	ACC_MEDIA_MOVEL 			:= 0;		//RESET DO ACUMULADOR DA MEDIA MOVEL
   	CONTAGEM					:= 0;		//RESET DO CONTADOR DE POSIÇAO DO VETOR
   	CALCULA_ALEATORIOS 			:= 0;		//RESET DO RANDOMIZADOR
   	DISSIPACAO					:= 0;
   	P_ENTRADA					:= 0;
   
   	//RESETA E DESLIGA O LOOP PID
   	TEMPO_LOOP_PID.RESET			:= 1;
   	TEMPO_LOOP_PID.ENABLEIN 		:= 0;
   	TEMPO_LOOP_PID.TIMERENABLE 		:= 0;
   
   	//RESETA E DESLIGA O SUAVIZADOR/ATRASADOR
   	TEMPO_MEDIA_MOVEL.RESET 		:= 1;
   	TEMPO_MEDIA_MOVEL.ENABLEIN 		:= 0;
   	TEMPO_MEDIA_MOVEL.TIMERENABLE 	:= 0;
   
   	//RESETA E DESLIGA O SISTEMA
   	TEMPO_LOOP_SISTEMA.RESET		:= 1;
   	TEMPO_LOOP_SISTEMA.ENABLEIN 	:= 0;
   	TEMPO_LOOP_SISTEMA.TIMERENABLE 	:= 0;
   
   END_IF;
   
   
   ////////////////////////////////////////////////////////////////////////////
   //							CONTROLE PID
   ////////////////////////////////////////////////////////////////////////////
   
   //TEMPO DO LOOP PID
   T_AMOST_PID :=	5*T_LOOP_SISTEMA;
   TEMPO_LOOP_PID.RESET := 0;
   TEMPO_LOOP_PID.ENABLEIN := 1;
   TEMPO_LOOP_PID.TIMERENABLE := 1;
   TEMPO_LOOP_PID.PRE := T_AMOST_PID;
   
   
   //CONVERSAO PARA SEGUNDOS EM FLOAT
   TIME_PID := T_AMOST_PID/1000;
   
   
   IF TEMPO_LOOP_PID.DN THEN
   
   	//CALCULO DO ERRO
   	ERRO := (SP - PV);
   
   	//CALCULO DA INTEGRAL
   	INTEGRAL := INTEGRAL + (ERRO*TIME_PID);
   
   	//LIMITES DA INTEGRAL
   	IF INTEGRAL > 100 THEN
   		INTEGRAL := 100;
   	END_IF;
   	IF INTEGRAL < -100 THEN
   		INTEGRAL := -100;
   	END_IF;
   
   	//EVITA O ERRO DE DIVISAO POR ZERO
   	IF TI <= 0 THEN
   		TI_INV := 0;
   	ELSE
   		TI_INV := 1/TI;
   	END_IF;
   
   	//CALCULO DA DERIVADA
   	DERIVADA := (ERRO - ERRO_ANTERIOR)/TIME_PID;
   
   	//CALCULO DA SAIDA O PID
   	ABERTURA_VALVULA := KP*(ERRO + TI_INV*INTEGRAL + TD*DERIVADA);
   
   	//ATUALIZA O ERRO ANTERIOR
   	ERRO_ANTERIOR := ERRO;
   
   	//LIMITA ABERTURA DA VALVULA
   	IF ABERTURA_VALVULA < 0 THEN
   		ABERTURA_VALVULA := 0;
   	END_IF;
   
   	IF ABERTURA_VALVULA > 100 THEN
   		ABERTURA_VALVULA := 100;
   	END_IF;
   
   	TEMPO_LOOP_PID.RESET := 1;
   
   END_IF;
   
   
   ////////////////////////////////////////////////////////////////////////////
   //						SIMULACAO DO CONSUMO
   ////////////////////////////////////////////////////////////////////////////
   
   
   IF NOT(CALCULA_ALEATORIOS) THEN
   
   	//SORTEIA UM TEMPO DE CONSUMO DE 0 A 5 SEGUNDOS
   	SEED := (12345*SEED + 12345)MOD(432);
   	ALEATORIO := SEED / 432;
   	TEMPO_CONSUMINDO.PRE := 5000*ALEATORIO;
   
   	//SORTEIA UM TEMPO SEM CONSUMIR DE 0 A 2 SEGUNDOS
   	SEED := (12345*SEED + 12345)MOD(432);
   	ALEATORIO := SEED / 432;
   	TEMPO_SEM_CONSUMO.PRE := 2000*ALEATORIO;
   
   	//SORTEIA UM VALOR PARA CONSUMO
   	SEED := (12345*SEED + 12345)MOD(432);
   	ALEATORIO := SEED / 432;
   	CONSUMO_ALEATORIO := (30000*ALEATORIO + 1)*(FATOR_CONSUMO/100);
   
   	//FINALIZA O CALCULO DE ALEATORIOS
   	CALCULA_ALEATORIOS := 1;
   
   END_IF;
   
   
   //ALTERNANDO OS TEMPORIZADORES DE CONSUMO
   IF CONSUMIR THEN
   
   	//RESETA O TEMPORIZADOR SEM CONSUMO
   	TEMPO_SEM_CONSUMO.RESET			:= 1;
   	TEMPO_SEM_CONSUMO.ENABLEIN		:= 0;
   	TEMPO_SEM_CONSUMO.TIMERENABLE	:= 0;
   
   	//APLICA O CONSUMO
   	CONSUMINDO := CONSUMO_ALEATORIO;
   
   	//LIGA O TIMER DE CONSUMO
   	TEMPO_CONSUMINDO.ENABLEIN 		:= 1;
   	TEMPO_CONSUMINDO.RESET	  		:= 0;
   	TEMPO_CONSUMINDO.TIMERENABLE 	:= 1;
   	IF TEMPO_CONSUMINDO.DN THEN
   		CONSUMIR := 0;
   	END_IF;
   
   ELSE
   
   	//RESETA O TEMPORIZADOR DE CONSUMO
   	TEMPO_CONSUMINDO.RESET	  		:= 1;
   	TEMPO_CONSUMINDO.ENABLEIN 		:= 0;
   	TEMPO_CONSUMINDO.TIMERENABLE 	:= 0;
   
   	//DESLIGA O CONSUMO
   	CONSUMINDO := 1;
   
   	//LIGA TEMPO SEM CONSUMIR
   	TEMPO_SEM_CONSUMO.ENABLEIN		:= 1;
   	TEMPO_SEM_CONSUMO.RESET			:= 0;
   	TEMPO_SEM_CONSUMO.TIMERENABLE	:= 1;
   
   	//REINICIA O CICLO
   	IF TEMPO_SEM_CONSUMO.DN THEN
   		CONSUMIR := 1;
   
   		//DISPARA UM NOVO CALCULO DE ALEATORIOS
   		CALCULA_ALEATORIOS := 0;
   
   	END_IF;
   
   END_IF;
   
   
   ////////////////////////////////////////////////////////////////////////////
   //		   SUAVIZAÇÃO E ATRASO DO SINAL DO SENSOR POR MEDIA MOVEL
   ////////////////////////////////////////////////////////////////////////////
   
   
   //LIGANDO O ATRASO/SUAVIZACAO
   IF ATRASO_SENSOR > 20 THEN
   
   	//ALOCA O BUFFER DE MEDIA MOVEL
   	TAMANHO_BUFFER := ATRASO_SENSOR/20;
   
   	//TEMPORIZADOR DE AMOSTRAGEM
   	TEMPO_MEDIA_MOVEL.RESET 		:= 0;
   	TEMPO_MEDIA_MOVEL.PRE 			:= 2*T_LOOP_SISTEMA;
   	TEMPO_MEDIA_MOVEL.ENABLEIN 		:= 1;
   	TEMPO_MEDIA_MOVEL.TIMERENABLE	:= 1;
   
   	//CONSIDERAMOS O TEMPO DE ATRASO COMO O TEMPO DA MEDIANA DOS DADOS AMOSTRADOS SALVOS NO VETOR
   	//ENTAO O ATRASO SERA: (N_DADOS*TEMPO_AMOSTRAGEM)/2
   
   	IF TEMPO_MEDIA_MOVEL.DN THEN
   
   		//LIGA O BUFFER CIRCULAR (VETOR CHEIO)
   		IF BUFFER_CIRCULAR THEN
   			//RETIRA O ULTIMO VALOR DO VETOR
   			ACC_MEDIA_MOVEL := ACC_MEDIA_MOVEL - VETOR_VALORES[CONTAGEM];
   		END_IF;
   
   		//ACUMULA OS K-ULTIMOS VALORES
   		ACC_MEDIA_MOVEL := ACC_MEDIA_MOVEL + P_SAIDA;
   
   		//ADICIONA O NOVO VALOR NA POSICAO DO ULTIMO RETIRADO
   		VETOR_VALORES[CONTAGEM] := P_SAIDA;
   
   		//INCREMENTA A POSICAO DO VETOR
   		CONTAGEM := CONTAGEM + 1;
   
   		//SE O VETOR ENCHEU, LIGA O BUFFER CIRCULAR E VOLTA AO SEU INICIO
   		IF CONTAGEM > TAMANHO_BUFFER-1 THEN
   			BUFFER_CIRCULAR :=1;
   			CONTAGEM := 0;
   		END_IF;
   
   		//RESET DO TEMPORIZADOR
   		TEMPO_MEDIA_MOVEL.RESET := 1;
   
   	END_IF;
   
   	//ATUALIZA O VALOR DO SENSOR DE PRESAO
   	PV := ACC_MEDIA_MOVEL/TAMANHO_BUFFER;
   
   ELSE
   
   	//SEM ATRASO
   	PV := P_SAIDA;
   
   END_IF;
   
   
   ////////////////////////////////////////////////////////////////FIM!!!
   
   
   
   
   
END_ROUTINE
END_PROGRAM
